FUNCTION_BLOCK MPC_MOVE_BLOCKED_NMPC_V3E (* Fail-closed delay-aware move-blocked nonlinear MPC V3 with 9 s AppliedDAC history and 500 ms execution period *)
  (* Standard: 61499-2 *)
  (* Version 3.0, 2026-08-18, Guilherme *)
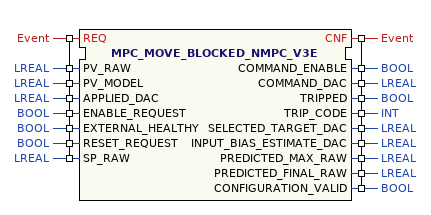
  EVENT_INPUT
    REQ WITH PV_RAW, PV_MODEL, APPLIED_DAC, ENABLE_REQUEST, EXTERNAL_HEALTHY, RESET_REQUEST, SP_RAW; (* Execute one 500 ms delay-aware MPC V3 cycle *)
  END_EVENT
  EVENT_OUTPUT
    CNF WITH COMMAND_ENABLE, COMMAND_DAC, TRIPPED, TRIP_CODE, SELECTED_TARGET_DAC, INPUT_BIAS_ESTIMATE_DAC, PREDICTED_MAX_RAW, PREDICTED_FINAL_RAW, CONFIGURATION_VALID; (* MPC cycle completed *)
  END_EVENT
  VAR_INPUT
    PV_RAW : LREAL; (* Unfiltered raw level used by the measured hard trip *)
    PV_MODEL : LREAL; (* 9-sample rolling-median raw level used by the identified model *)
    APPLIED_DAC : LREAL; (* PLC-confirmed DAC used as the move-constraint reference *)
    ENABLE_REQUEST : BOOL; (* Explicit operator/commissioning enable; FALSE is normal zero-output mode *)
    EXTERNAL_HEALTHY : BOOL; (* PLC/gateway watchdog healthy input *)
    RESET_REQUEST : BOOL; (* Explicitly clear the latched MPC trip and internal estimator state *)
    SP_RAW : LREAL; (* Raw-count setpoint; first commissioning value is 450 *)
  END_VAR
  VAR_OUTPUT
    COMMAND_ENABLE : BOOL; (* Fail-closed actuator enable request *)
    COMMAND_DAC : LREAL; (* MPC DAC request before downstream defense-in-depth limiting *)
    TRIPPED : BOOL; (* Latched MPC trip state *)
    TRIP_CODE : INT; (* 0=none,1=health,2=PV invalid,3=measured high,4=AppliedDAC,5=setpoint,6=no feasible prediction *)
    SELECTED_TARGET_DAC : LREAL; (* Move-blocked target selected by the current horizon search *)
    INPUT_BIAS_ESTIMATE_DAC : LREAL; (* Bounded offset-compensation estimate *)
    PREDICTED_MAX_RAW : LREAL; (* Maximum predicted model level for the selected candidate *)
    PREDICTED_FINAL_RAW : LREAL; (* Final horizon model level for the selected candidate *)
    CONFIGURATION_VALID : BOOL; (* Frozen V1 commissioning configuration is internally valid *)
  END_VAR
  VAR
    trip_latched_internal : BOOL := FALSE;
    trip_code_internal : INT := 0;
    history_count : DINT := 0;
    record_history_internal : BOOL := FALSE;
    best_found : BOOL := FALSE;
    candidate_feasible : BOOL := FALSE;
    h00 : LREAL := 0.0;
    h01 : LREAL := 0.0;
    h02 : LREAL := 0.0;
    h03 : LREAL := 0.0;
    h04 : LREAL := 0.0;
    h05 : LREAL := 0.0;
    h06 : LREAL := 0.0;
    h07 : LREAL := 0.0;
    h08 : LREAL := 0.0;
    h09 : LREAL := 0.0;
    h10 : LREAL := 0.0;
    h11 : LREAL := 0.0;
    h12 : LREAL := 0.0;
    h13 : LREAL := 0.0;
    h14 : LREAL := 0.0;
    h15 : LREAL := 0.0;
    h16 : LREAL := 0.0;
    h17 : LREAL := 0.0;
    q00 : LREAL := 0.0;
    q01 : LREAL := 0.0;
    q02 : LREAL := 0.0;
    q03 : LREAL := 0.0;
    q04 : LREAL := 0.0;
    q05 : LREAL := 0.0;
    q06 : LREAL := 0.0;
    q07 : LREAL := 0.0;
    q08 : LREAL := 0.0;
    q09 : LREAL := 0.0;
    q10 : LREAL := 0.0;
    q11 : LREAL := 0.0;
    q12 : LREAL := 0.0;
    q13 : LREAL := 0.0;
    q14 : LREAL := 0.0;
    q15 : LREAL := 0.0;
    q16 : LREAL := 0.0;
    q17 : LREAL := 0.0;
    best_cost : LREAL := 0.0;
    best_target : LREAL := 0.0;
    best_predicted_max : LREAL := 0.0;
    best_predicted_final : LREAL := 0.0;
    candidate_target : LREAL := 0.0;
    predicted_y : LREAL := 0.0;
    predicted_u : LREAL := 0.0;
    previous_u : LREAL := 0.0;
    delayed_u : LREAL := 0.0;
    candidate_cost : LREAL := 0.0;
    candidate_predicted_max : LREAL := 0.0;
    delta_u : LREAL := 0.0;
    effective_input : LREAL := 0.0;
    phi_value : LREAL := 0.0;
    tracking_error : LREAL := 0.0;
    move_value : LREAL := 0.0;
    soft_excess : LREAL := 0.0;
    terminal_error : LREAL := 0.0;
    command_candidate : LREAL := 0.0;
    candidate_index : DINT := 0;
    prediction_index : DINT := 0;
  END_VAR
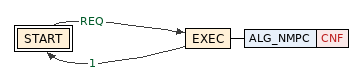
  EC_STATES
    START;
    EXEC : ALG_NMPC -> CNF;
  END_STATES
  EC_TRANSITIONS
    START TO EXEC := REQ;
    EXEC TO START := 1;
  END_TRANSITIONS
  ALGORITHM ALG_NMPC IN ST: (* Frozen move-blocked NMPC V1 with model constraints, trip latch, offset compensation, and piecewise-linear x^1.2 model input *)
IF RESET_REQUEST THEN
    trip_latched_internal := FALSE;
    trip_code_internal := 0;
END_IF;

CONFIGURATION_VALID := TRUE;
COMMAND_ENABLE := FALSE;
COMMAND_DAC := LREAL#0.0;
SELECTED_TARGET_DAC := LREAL#0.0;
INPUT_BIAS_ESTIMATE_DAC := LREAL#0.0;
PREDICTED_MAX_RAW := LREAL#-1.0;
PREDICTED_FINAL_RAW := LREAL#-1.0;

record_history_internal := (PV_RAW = PV_RAW) AND (PV_MODEL = PV_MODEL) AND (APPLIED_DAC = APPLIED_DAC) AND (SP_RAW = SP_RAW) AND (APPLIED_DAC >= LREAL#0.0) AND (APPLIED_DAC <= LREAL#12000.0);

IF NOT trip_latched_internal THEN
    IF NOT ENABLE_REQUEST THEN
        COMMAND_ENABLE := FALSE;
        COMMAND_DAC := LREAL#0.0;
    ELSE
        IF NOT EXTERNAL_HEALTHY THEN
            trip_latched_internal := TRUE;
            trip_code_internal := 2;
        ELSIF NOT (PV_RAW = PV_RAW) OR NOT (PV_MODEL = PV_MODEL) OR NOT (APPLIED_DAC = APPLIED_DAC) OR NOT (SP_RAW = SP_RAW) THEN
            trip_latched_internal := TRUE;
            trip_code_internal := 1;
        ELSIF PV_RAW < LREAL#0.0 OR PV_MODEL < LREAL#0.0 OR PV_RAW >= LREAL#1500.0 THEN
            trip_latched_internal := TRUE;
            trip_code_internal := 3;
        ELSIF APPLIED_DAC < LREAL#0.0 OR APPLIED_DAC > LREAL#12000.0 THEN
            trip_latched_internal := TRUE;
            trip_code_internal := 4;
        ELSIF SP_RAW < LREAL#0.0 OR SP_RAW >= LREAL#800.0 THEN
            trip_latched_internal := TRUE;
            trip_code_internal := 5;
        ELSIF history_count < 18 THEN
            trip_latched_internal := TRUE;
            trip_code_internal := 7;
        ELSE
            best_found := FALSE;
            best_cost := LREAL#1000000000.0;
            best_target := LREAL#0.0;
            best_predicted_max := LREAL#-1.0;
            best_predicted_final := LREAL#-1.0;
            FOR candidate_index := 0 TO 12 DO
                CASE candidate_index OF
                    0:
                        candidate_target := LREAL#0.0;
                    1:
                        candidate_target := LREAL#11500.0;
                    2:
                        candidate_target := LREAL#11550.0;
                    3:
                        candidate_target := LREAL#11600.0;
                    4:
                        candidate_target := LREAL#11650.0;
                    5:
                        candidate_target := LREAL#11700.0;
                    6:
                        candidate_target := LREAL#11750.0;
                    7:
                        candidate_target := LREAL#11800.0;
                    8:
                        candidate_target := LREAL#11845.626677302696407;
                    9:
                        candidate_target := LREAL#11850.0;
                    10:
                        candidate_target := LREAL#11900.0;
                    11:
                        candidate_target := LREAL#11950.0;
                    12:
                        candidate_target := LREAL#12000.0;
                    ELSE
                        candidate_target := LREAL#0.0;
                END_CASE;
                q00 := h00;
                q01 := h01;
                q02 := h02;
                q03 := h03;
                q04 := h04;
                q05 := h05;
                q06 := h06;
                q07 := h07;
                q08 := h08;
                q09 := h09;
                q10 := h10;
                q11 := h11;
                q12 := h12;
                q13 := h13;
                q14 := h14;
                q15 := h15;
                q16 := h16;
                q17 := h17;
                IF PV_MODEL < LREAL#288.0 THEN
                    predicted_y := LREAL#288.0;
                ELSE
                    predicted_y := PV_MODEL;
                END_IF;
                predicted_u := APPLIED_DAC;
                previous_u := APPLIED_DAC;
                candidate_cost := LREAL#0.0;
                candidate_predicted_max := predicted_y;
                candidate_feasible := TRUE;
                FOR prediction_index := 1 TO 60 DO
                    IF candidate_feasible THEN
                        delta_u := candidate_target - predicted_u;
                        IF delta_u > LREAL#750.0 THEN
                            delta_u := LREAL#750.0;
                        ELSIF delta_u < LREAL#-750.0 THEN
                            delta_u := LREAL#-750.0;
                        END_IF;
                        predicted_u := predicted_u + delta_u;
                        IF predicted_u > LREAL#12000.0 THEN
                            predicted_u := LREAL#12000.0;
                        ELSIF predicted_u < LREAL#0.0 THEN
                            predicted_u := LREAL#0.0;
                        END_IF;
                        delayed_u := q00;
                        q00 := q01;
                        q01 := q02;
                        q02 := q03;
                        q03 := q04;
                        q04 := q05;
                        q05 := q06;
                        q06 := q07;
                        q07 := q08;
                        q08 := q09;
                        q09 := q10;
                        q10 := q11;
                        q11 := q12;
                        q12 := q13;
                        q13 := q14;
                        q14 := q15;
                        q15 := q16;
                        q16 := q17;
                        q17 := predicted_u;
                        effective_input := delayed_u - LREAL#11750.0;
                        IF effective_input < LREAL#0.0 THEN
                            effective_input := LREAL#0.0;
                        ELSIF effective_input > LREAL#500.0 THEN
                            effective_input := LREAL#500.0;
                        END_IF;
                        IF effective_input <= LREAL#0.0 THEN
                            phi_value := LREAL#0.0;
                        ELSIF effective_input <= LREAL#50.0 THEN
                            phi_value := LREAL#0.0 + LREAL#2.186724147886556 * (effective_input - LREAL#0.0);
                        ELSIF effective_input <= LREAL#100.0 THEN
                            phi_value := LREAL#109.336207394327786 + LREAL#2.837048715132604 * (effective_input - LREAL#50.0);
                        ELSIF effective_input <= LREAL#150.0 THEN
                            phi_value := LREAL#251.188643150957972 + LREAL#3.148436919260821 * (effective_input - LREAL#100.0);
                        ELSIF effective_input <= LREAL#200.0 THEN
                            phi_value := LREAL#408.610489113999051 + LREAL#3.369389464977726 * (effective_input - LREAL#150.0);
                        ELSIF effective_input <= LREAL#250.0 THEN
                            phi_value := LREAL#577.07996236288534 + LREAL#3.543841594105197 * (effective_input - LREAL#200.0);
                        ELSIF effective_input <= LREAL#300.0 THEN
                            phi_value := LREAL#754.272042068145197 + LREAL#3.689367025828481 * (effective_input - LREAL#250.0);
                        ELSIF effective_input <= LREAL#350.0 THEN
                            phi_value := LREAL#938.740393359569225 + LREAL#3.814953797640478 * (effective_input - LREAL#300.0);
                        ELSIF effective_input <= LREAL#400.0 THEN
                            phi_value := LREAL#1129.488083241593131 + LREAL#3.925870473888026 * (effective_input - LREAL#350.0);
                        ELSIF effective_input <= LREAL#450.0 THEN
                            phi_value := LREAL#1325.781606935994432 + LREAL#4.025491573724398 * (effective_input - LREAL#400.0);
                        ELSIF effective_input <= LREAL#500.0 THEN
                            phi_value := LREAL#1527.056185622214343 + LREAL#4.116118445313023 * (effective_input - LREAL#450.0);
                        ELSE
                            phi_value := LREAL#1732.862107887865477;
                        END_IF;
                        predicted_y := LREAL#288.0 + LREAL#0.900087626252259 * (predicted_y - LREAL#288.0) + LREAL#0.067989118863552 * phi_value;
                        IF predicted_y > candidate_predicted_max THEN
                            candidate_predicted_max := predicted_y;
                        END_IF;
                        IF NOT (predicted_y = predicted_y) OR predicted_y > LREAL#1400.0 THEN
                            candidate_feasible := FALSE;
                        ELSE
                            tracking_error := predicted_y - SP_RAW;
                            move_value := predicted_u - previous_u;
                            candidate_cost := candidate_cost + LREAL#5.0 * tracking_error * tracking_error + LREAL#0.00004 * move_value * move_value;
                            IF predicted_y > LREAL#1100.0 THEN
                                soft_excess := predicted_y - LREAL#650.0;
                                candidate_cost := candidate_cost + LREAL#100.0 * soft_excess * soft_excess;
                            END_IF;
                            previous_u := predicted_u;
                        END_IF;
                    END_IF;
                END_FOR;
                IF candidate_feasible THEN
                    terminal_error := predicted_y - SP_RAW;
                    candidate_cost := candidate_cost + LREAL#10.0 * terminal_error * terminal_error;
                    IF (NOT best_found) OR candidate_cost < best_cost THEN
                        best_found := TRUE;
                        best_cost := candidate_cost;
                        best_target := candidate_target;
                        best_predicted_max := candidate_predicted_max;
                        best_predicted_final := predicted_y;
                    END_IF;
                END_IF;
            END_FOR;
            IF NOT best_found THEN
                trip_latched_internal := TRUE;
                trip_code_internal := 6;
            ELSE
                delta_u := best_target - APPLIED_DAC;
                IF delta_u > LREAL#750.0 THEN
                    delta_u := LREAL#750.0;
                ELSIF delta_u < LREAL#-750.0 THEN
                    delta_u := LREAL#-750.0;
                END_IF;
                command_candidate := APPLIED_DAC + delta_u;
                IF command_candidate > LREAL#12000.0 THEN
                    command_candidate := LREAL#12000.0;
                ELSIF command_candidate < LREAL#0.0 THEN
                    command_candidate := LREAL#0.0;
                END_IF;
                COMMAND_ENABLE := TRUE;
                COMMAND_DAC := command_candidate;
                SELECTED_TARGET_DAC := best_target;
                PREDICTED_MAX_RAW := best_predicted_max;
                PREDICTED_FINAL_RAW := best_predicted_final;
            END_IF;
        END_IF;
    END_IF;
END_IF;

IF record_history_internal THEN
    h00 := h01;
    h01 := h02;
    h02 := h03;
    h03 := h04;
    h04 := h05;
    h05 := h06;
    h06 := h07;
    h07 := h08;
    h08 := h09;
    h09 := h10;
    h10 := h11;
    h11 := h12;
    h12 := h13;
    h13 := h14;
    h14 := h15;
    h15 := h16;
    h16 := h17;
    h17 := APPLIED_DAC;
    IF history_count < 18 THEN
        history_count := history_count + 1;
    END_IF;
END_IF;

TRIPPED := trip_latched_internal;
TRIP_CODE := trip_code_internal;
INPUT_BIAS_ESTIMATE_DAC := LREAL#0.0;

IF trip_latched_internal THEN
    COMMAND_ENABLE := FALSE;
    COMMAND_DAC := LREAL#0.0;
    SELECTED_TARGET_DAC := LREAL#0.0;
    PREDICTED_MAX_RAW := LREAL#-1.0;
    PREDICTED_FINAL_RAW := LREAL#-1.0;
END_IF;
  END_ALGORITHM
END_FUNCTION_BLOCK
